FUNCTION F_ClearMem : BOOL
VAR_INPUT
    Data : ANY;
END_VAR
VAR
END_VAR

MEMSET(
    destAddr := Data.pValue,
    fillByte := 0,
    n        := DINT_TO_UDINT(Data.diSize));

END_FUNCTION

(* stored: Version 1.1.0.1, ProductVersion 3.1.4024.3
   POU F_ClearMem: Id {2b5ec06a-09fa-07e4-19a0-d175ac60f6b4}, SpecialFunc None *)
